FUNCTION_BLOCK FB_Handheld
VAR_INPUT
END_VAR
VAR_OUTPUT
	fbVorTrig:				R_TRIG;
	fbZurueckTrig:			R_TRIG;
	nGewaehlteStation:		INT;
END_VAR
VAR
	bE_TasteVor				AT%I*:	BOOL;
	bE_TasteZurueck			AT%I*:	BOOL;
	bE_Zustimmtaster		AT%I*:	BOOL;
	
	bA_LampeHandheld		AT%Q*:	BOOL;
END_VAR

//********************************************************************************
//Handheld
fbVorTrig(CLK := bE_TasteVor AND bE_Zustimmtaster);
fbZurueckTrig(CLK := bE_TasteZurueck AND bE_Zustimmtaster);

bA_LampeHandheld := bE_Zustimmtaster AND MAIN.bE_Handbetrieb;

END_FUNCTION_BLOCK

(* stored: Version 1.1.0.1, ProductVersion 3.1.4024.12
   POU FB_Handheld: Id {5c525b99-8183-47d7-83a4-ced87fc372b9}, SpecialFunc None *)
